FUNCTION ConcatArray : T_MaxString
VAR_INPUT
	sArrExpressions: ARRAY[0..15] OF T_maxString;
END_VAR
VAR
	ii: INT;
END_VAR

ConcatArray := '';

FOR ii:=0 TO 15 DO
	ConcatArray := CONCAT(ConcatArray, sArrExpressions[ii]);
END_FOR

END_FUNCTION

(* stored: Version 1.1.0.1
   POU ConcatArray: Id {2b444c08-fa69-41e5-9ca7-682b0db83e98}, SpecialFunc None *)
